TYPE ST_DebugColumnAIO :
STRUCT
END_STRUCT
END_TYPE

(* stored: Version 1.1.0.1, ProductVersion 3.1.4022.18
   DUT ST_DebugColumnAIO: Id {65f0873b-b25f-4117-8d71-16802f68f1c6} *)
